(* PLC project Unnamed, Unknown Unnamed 1 *)
(* stored: creationDateTime 2025-11-14T15:23:30, modificationDateTime 2026-02-02T00:07:13 *)

PROGRAM program0
  VAR
    Start : BOOL;
    Stop : BOOL;
    CycleOn : BOOL;
    InletValve : BOOL;
    LevelSensor2 : BOOL;
    Valve2 : BOOL;
    TempSensor1 : INT := 59;
    TempSensor2 : INT := 12;
    OutletValve1 : BOOL;
    OutletValve2 : BOOL;
    Heater : BOOL;
    LevelSensor4 : BOOL;
    LevelSensor1 : BOOL;
    LevelSensor3 : BOOL;
    Valve3 : BOOL;
    Cooler : BOOL;
  END_VAR

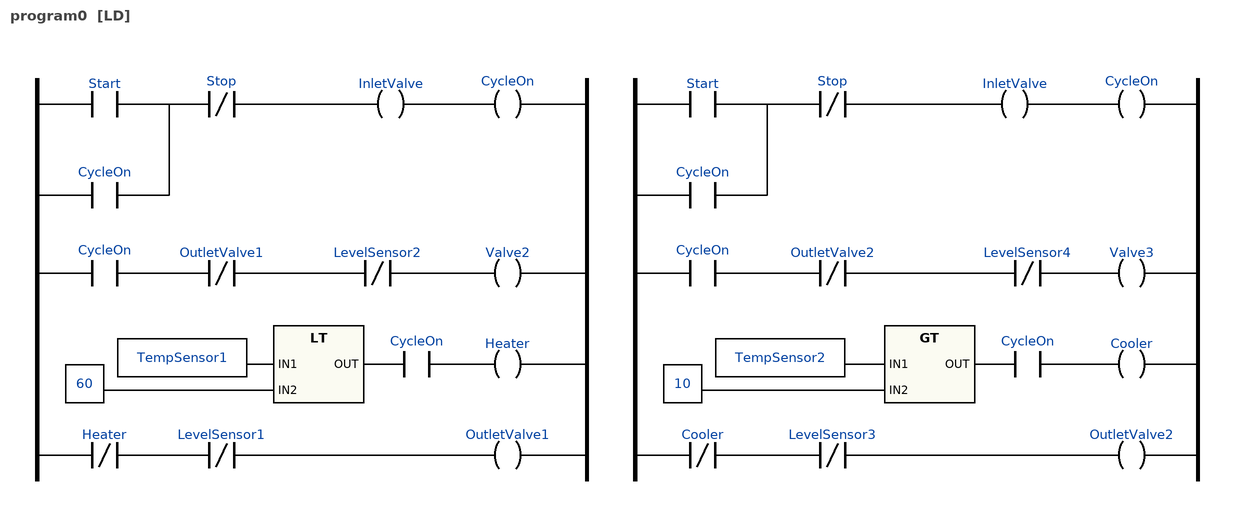
(* LD diagram, written out as Structured Text *)
CycleOn := (Start OR CycleOn) AND NOT Stop;
InletValve := (Start OR CycleOn) AND NOT Stop;
Valve2 := CycleOn AND NOT OutletValve1 AND NOT LevelSensor2;
Heater := TempSensor1 < 60 AND CycleOn;
OutletValve1 := NOT Heater AND NOT LevelSensor1;
CycleOn := (Start OR CycleOn) AND NOT Stop;
InletValve := (Start OR CycleOn) AND NOT Stop;
Valve3 := CycleOn AND NOT OutletValve2 AND NOT LevelSensor4;
Cooler := TempSensor2 > 10 AND CycleOn;
OutletValve2 := NOT Cooler AND NOT LevelSensor3;
END_PROGRAM

CONFIGURATION Config0
  RESOURCE Res0 ON PLC
    TASK task0(INTERVAL := T#20ms, PRIORITY := 0);
    PROGRAM instance0 WITH task0 : program0;
  END_RESOURCE
END_CONFIGURATION
